// TIA Portal V19 export
TYPE "PPrf_A0304_0304_Scarico"
// stored: Access Published
   STRUCT
      Trasporto : "PPrf_A0303_Trasporto";
      Navetta : "PPrf_A0304_Navetta";
   END_STRUCT;
END_TYPE
